FUNCTION_BLOCK fb_xmeas_acquire

VAR_INPUT
END_VAR

VAR_OUTPUT
END_VAR

VAR
END_VAR

END_FUNCTION_BLOCK

(* stored: Version 1.1.0.1, ProductVersion 3.1.0.26
   POU fb_xmeas_acquire: Id {cd0e3f91-bbf0-4630-b6d2-13bb1b3d09c9} *)
